{attribute 'GeneratedUsingTerminal: IODEVICETYPE_ETHERCATPROT'}
{attribute addProperty BoxType "IODEVICETYPE_ETHERCATPROT"}
{attribute addProperty Id "R2_EK1100R2_EK1100_DD939EB7488R3_EK1100R3_EK1100_0213442E786R4_EK1100R4_EK1100_717E66DB159R5_EK1100R5_EK1100_F6AE5C4E553R6_EK1100R6_EK1100_AAF8B27B344R6_1_EK1100R6_1_EK1100_E0142E79442R7_EK1100R7_EK1100_541C839D286SyncUnitsSyncUnits_03D3E917360InputsInputs_A65FACA410OutputsOutputs_23C0ED1D6InfoDataInfoData_84133AC922"}
{attribute addProperty CRC "2215286339"}
{attribute addProperty Size "3456"}
TYPE _2100260_A1_LAN_0_R2_840A9643 :
STRUCT
	{attribute addProperty Name "R2_EK1100"}
	{attribute addProperty PreviousPort "2100260_A1_LAN_0_R2 : Master"}
	R2_EK1100 : R2_EK1100_DD939EB7;
	{attribute addProperty Name "R3_EK1100"}
	{attribute addProperty PreviousPort "R2 (EK1100) : C"}
	R3_EK1100 : R3_EK1100_0213442E;
	{attribute addProperty Name "R4_EK1100"}
	{attribute addProperty PreviousPort "R3 (EK1100) : C"}
	R4_EK1100 : R4_EK1100_717E66DB;
	{attribute addProperty Name "R5_EK1100"}
	{attribute addProperty PreviousPort "R4 (EK1100) : C"}
	R5_EK1100 : R5_EK1100_F6AE5C4E;
	{attribute addProperty Name "R6_EK1100"}
	{attribute addProperty PreviousPort "R5 (EK1100) : C"}
	R6_EK1100 : R6_EK1100_AAF8B27B;
	{attribute addProperty Name "R6_1_EK1100"}
	{attribute addProperty PreviousPort "R6 (EK1100) : C"}
	R6_1_EK1100 : R6_1_EK1100_E0142E79;
	{attribute addProperty Name "R7_EK1100"}
	{attribute addProperty PreviousPort "R6_1 (EK1100) : C"}
	R7_EK1100 : R7_EK1100_541C839D;
	{attribute addProperty Name "SyncUnits"}
	SyncUnits : SyncUnits_03D3E917;
	{attribute addProperty Name "Inputs"}
	Inputs : TcoIo.Inputs_A65FACA4;
	{attribute addProperty Name "Outputs"}
	Outputs : TcoIo.Outputs_23C0ED1D;
	{attribute addProperty Name "InfoData"}
	InfoData : TcoIo.InfoData_84133AC9;
END_STRUCT
END_TYPE

(* stored: Version 1.2.0.0, ProductVersion 3.1.4024.9
   DUT _2100260_A1_LAN_0_R2_840A9643: Id {df433366-27bd-01a5-1092-a2ebca35be55} *)
